// TIA Portal V20 export
TYPE "UDT_Service_IndexElement"
   STRUCT
      startIndex : Int := -1;   // Start index for addressing parameter
      endIndex : Int := -1;   // End index for addressing parameter
   END_STRUCT;
END_TYPE
